# EPICS substitutions: MC07/MC07/tpmacApp/Db/pmacStatus.substitutions
file "db/pmacStatus.db"
{
pattern
{SYS,             PMAC,    VERSION  PLC  PORT,  NAXES }
{"XF:07ID1-OP",   "MC:07", "1"      5    "P0",  8     }
}
